// TIA Portal V19 export
FUNCTION "RECIRCULATION" : Void   // FC16, LAD
{ S7_Optimized_Access := 'TRUE' }
// stored: SetENOAutomatically false
BEGIN

REGION Network 1: MFG RECIRCULATION START
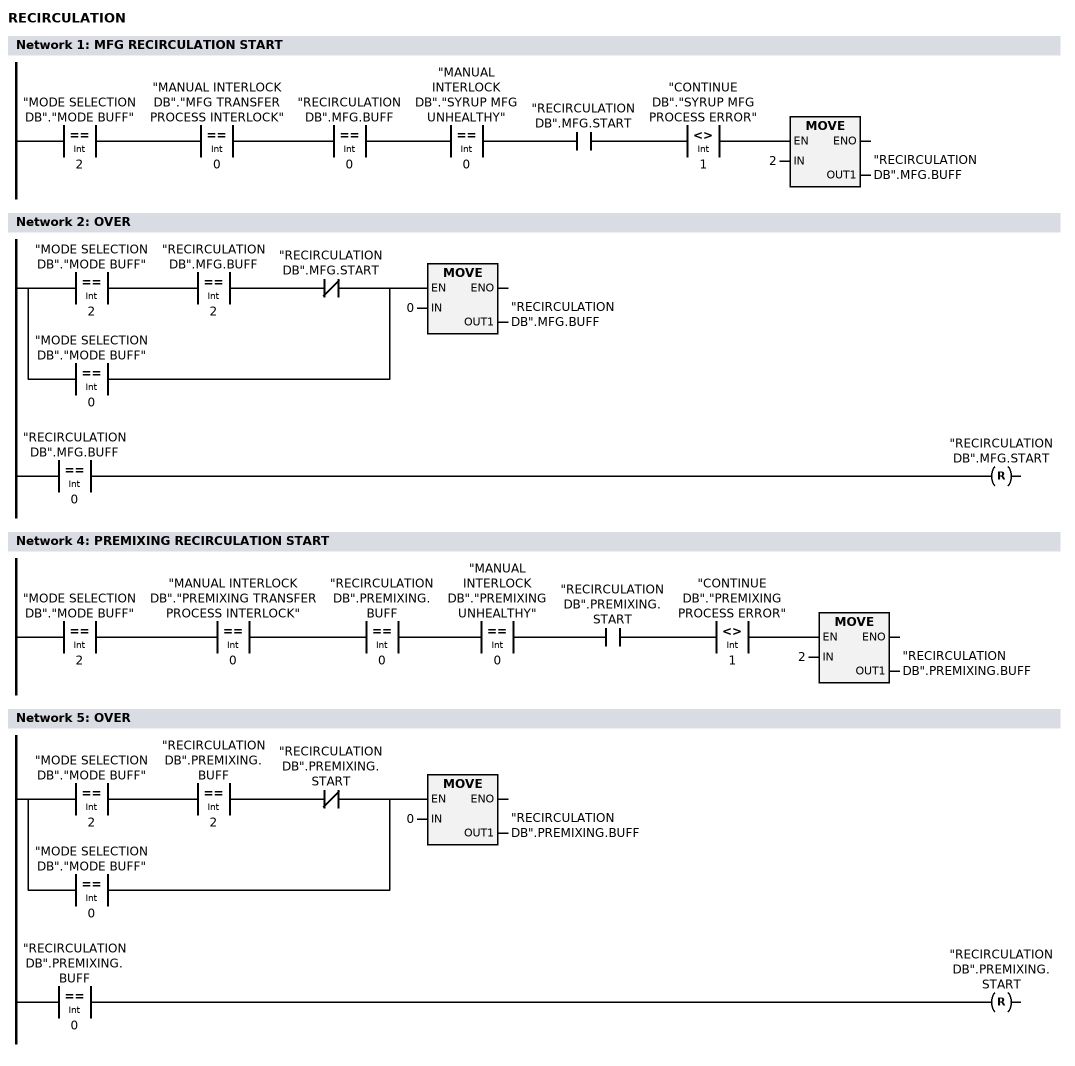
   RUNG wire#powerrail
      { S7_Templates := "SrcType := Int" } EQ_Contact(in1 := "MODE SELECTION DB"."MODE BUFF", in2 := 2)
      { S7_Templates := "SrcType := Int" } EQ_Contact(in1 := "MANUAL INTERLOCK DB"."MFG TRANSFER PROCESS INTERLOCK", in2 := 0)
      { S7_Templates := "SrcType := Int" } EQ_Contact(in1 := "RECIRCULATION DB".MFG.BUFF, in2 := 0)
      { S7_Templates := "SrcType := Int" } EQ_Contact(in1 := "MANUAL INTERLOCK DB"."SYRUP MFG UNHEALTHY", in2 := 0)
      Contact( "RECIRCULATION DB".MFG.START )
      { S7_Templates := "SrcType := Int" } NE_Contact(in1 := "CONTINUE DB"."SYRUP MFG PROCESS ERROR", in2 := 1)
      Move(in := 2, out1 => "RECIRCULATION DB".MFG.BUFF)
   END_RUNG
   // the same network as SCL:
   IF ("MODE SELECTION DB"."MODE BUFF" = 2) AND ("MANUAL INTERLOCK DB"."MFG TRANSFER PROCESS INTERLOCK" = 0) AND ("RECIRCULATION DB".MFG.BUFF = 0) AND ("MANUAL INTERLOCK DB"."SYRUP MFG UNHEALTHY" = 0) AND "RECIRCULATION DB".MFG.START AND ("CONTINUE DB"."SYRUP MFG PROCESS ERROR" <> 1) THEN
       "RECIRCULATION DB".MFG.BUFF := 2;
   END_IF;
END_REGION

REGION Network 2: OVER
   RUNG wire#powerrail
      { S7_Templates := "SrcType := Int" } EQ_Contact(in1 := "MODE SELECTION DB"."MODE BUFF", in2 := 2)
      { S7_Templates := "SrcType := Int" } EQ_Contact(in1 := "RECIRCULATION DB".MFG.BUFF, in2 := 2)
      I_Contact( "RECIRCULATION DB".MFG.START )
      wire#w1
      Move(in := 0, out1 => "RECIRCULATION DB".MFG.BUFF)
   END_RUNG
   RUNG wire#powerrail
      { S7_Templates := "SrcType := Int" } EQ_Contact(in1 := "MODE SELECTION DB"."MODE BUFF", in2 := 0)
   END_RUNG wire#w1
   RUNG wire#powerrail
      { S7_Templates := "SrcType := Int" } EQ_Contact(in1 := "RECIRCULATION DB".MFG.BUFF, in2 := 0)
      R_Coil( "RECIRCULATION DB".MFG.START )
   END_RUNG
   // the same network as SCL:
   IF (("MODE SELECTION DB"."MODE BUFF" = 2) AND ("RECIRCULATION DB".MFG.BUFF = 2) AND NOT "RECIRCULATION DB".MFG.START) OR ("MODE SELECTION DB"."MODE BUFF" = 0) THEN
       "RECIRCULATION DB".MFG.BUFF := 0;
   END_IF;
   IF "RECIRCULATION DB".MFG.BUFF = 0 THEN "RECIRCULATION DB".MFG.START := FALSE; END_IF;
END_REGION

REGION Network 4: PREMIXING RECIRCULATION START
   RUNG wire#powerrail
      { S7_Templates := "SrcType := Int" } EQ_Contact(in1 := "MODE SELECTION DB"."MODE BUFF", in2 := 2)
      { S7_Templates := "SrcType := Int" } EQ_Contact(in1 := "MANUAL INTERLOCK DB"."PREMIXING TRANSFER PROCESS INTERLOCK", in2 := 0)
      { S7_Templates := "SrcType := Int" } EQ_Contact(in1 := "RECIRCULATION DB".PREMIXING.BUFF, in2 := 0)
      { S7_Templates := "SrcType := Int" } EQ_Contact(in1 := "MANUAL INTERLOCK DB"."PREMIXING UNHEALTHY", in2 := 0)
      Contact( "RECIRCULATION DB".PREMIXING.START )
      { S7_Templates := "SrcType := Int" } NE_Contact(in1 := "CONTINUE DB"."PREMIXING PROCESS ERROR", in2 := 1)
      Move(in := 2, out1 => "RECIRCULATION DB".PREMIXING.BUFF)
   END_RUNG
   // the same network as SCL:
   IF ("MODE SELECTION DB"."MODE BUFF" = 2) AND ("MANUAL INTERLOCK DB"."PREMIXING TRANSFER PROCESS INTERLOCK" = 0) AND ("RECIRCULATION DB".PREMIXING.BUFF = 0) AND ("MANUAL INTERLOCK DB"."PREMIXING UNHEALTHY" = 0) AND "RECIRCULATION DB".PREMIXING.START AND ("CONTINUE DB"."PREMIXING PROCESS ERROR" <> 1) THEN
       "RECIRCULATION DB".PREMIXING.BUFF := 2;
   END_IF;
END_REGION

REGION Network 5: OVER
   RUNG wire#powerrail
      { S7_Templates := "SrcType := Int" } EQ_Contact(in1 := "MODE SELECTION DB"."MODE BUFF", in2 := 2)
      { S7_Templates := "SrcType := Int" } EQ_Contact(in1 := "RECIRCULATION DB".PREMIXING.BUFF, in2 := 2)
      I_Contact( "RECIRCULATION DB".PREMIXING.START )
      wire#w1
      Move(in := 0, out1 => "RECIRCULATION DB".PREMIXING.BUFF)
   END_RUNG
   RUNG wire#powerrail
      { S7_Templates := "SrcType := Int" } EQ_Contact(in1 := "MODE SELECTION DB"."MODE BUFF", in2 := 0)
   END_RUNG wire#w1
   RUNG wire#powerrail
      { S7_Templates := "SrcType := Int" } EQ_Contact(in1 := "RECIRCULATION DB".PREMIXING.BUFF, in2 := 0)
      R_Coil( "RECIRCULATION DB".PREMIXING.START )
   END_RUNG
   // the same network as SCL:
   IF (("MODE SELECTION DB"."MODE BUFF" = 2) AND ("RECIRCULATION DB".PREMIXING.BUFF = 2) AND NOT "RECIRCULATION DB".PREMIXING.START) OR ("MODE SELECTION DB"."MODE BUFF" = 0) THEN
       "RECIRCULATION DB".PREMIXING.BUFF := 0;
   END_IF;
   IF "RECIRCULATION DB".PREMIXING.BUFF = 0 THEN "RECIRCULATION DB".PREMIXING.START := FALSE; END_IF;
END_REGION
END_FUNCTION
